# EPICS IOC start-up script: iocBoot/iocxxx/examples/vme.iocsh
# BEGIN vme.cmd ---------------------------------------------------------------

### Scalers: Joerger VSC8/16
#dbLoadRecords("$(SCALER)/db/scaler.db","P=$(PREFIX),S=scaler2,OUT=#C1 S0 @,DTYP=Joerger VSC8/16,FREQ=10000000")
#- scaler database with modified calcs (user calcs for all 16 channels)
dbLoadRecords("$(SCALER)/db/scaler16m.db","P=$(PREFIX),S=scaler1,OUT=#C0 S0 @,DTYP=Joerger VSC8/16,FREQ=10000000")
#- Joerger VSC setup parameters:
#-     (1)cards, (2)base address(ext, 256-byte boundary),
#-     (3)interrupt vector (0=disable or  64 - 255)
VSCSetup(2, 0xB0000000, 200)

#- Joerger VS
#- scalerVS_Setup(int num_cards, /* maximum number of cards in crate */
#-       char *addrs,            /* address (0x800-0xf800, 2048-byte (0x800) boundary) */
#-       unsigned vector,        /* valid vectors(64-255) */
#-       int intlevel)
#scalerVS_Setup(1, 0x2000, 205, 5)
#epicsEnvSet("devScaler_VSDebug", 0)
#dbLoadRecords("$(STD)/stdApp/Db/scaler16m.db","P=$(PREFIX),S=scaler3,OUT=#C0 S0 @, DTYP=Joerger VS, FREQ=10000000")

# Heidenhain IK320 VME encoder interpolator
#dbLoadRecords("$(VME)/vmeApp/Db/IK320card.db","P=$(PREFIX),sw2=card0:,axis=1,switches=41344,irq=3")
#dbLoadRecords("$(VME)/vmeApp/Db/IK320card.db","P=$(PREFIX),sw2=card0:,axis=2,switches=41344,irq=3")
#dbLoadRecords("$(VME)/vmeApp/Db/IK320group.db","P=$(PREFIX),group=5")

# Struck 3801 MCS setup. mca 7-3-1
#< st_SIS3801.iocsh

# Struck 3820 MCS setup. mca 7-3-1
#< st_SIS3820.iocsh

#- VMI4116 setup parameters:
#-     (1)cards, (2)base address(short, 36-byte boundary),
#devAoVMI4116Debug = 20
#VMI4116_setup(1, 0xff00)
#dbLoadRecords("$(VME)/vmeApp/Db/VME_DAC.db", "P=$(PREFIX),D=2,C=0,N=1,S=0,DTYP=VMIVME-4116,H=65536,L=0", std)
#dbLoadRecords("$(VME)/vmeApp/Db/VME_DAC.db", "P=$(PREFIX),D=2,C=0,N=2,S=1,DTYP=VMIVME-4116,H=65536,L=0", std)
#dbLoadRecords("$(VME)/vmeApp/Db/VME_DAC.db", "P=$(PREFIX),D=2,C=0,N=3,S=2,DTYP=VMIVME-4116,H=65536,L=0", std)
#dbLoadRecords("$(VME)/vmeApp/Db/VME_DAC.db", "P=$(PREFIX),D=2,C=0,N=4,S=3,DTYP=VMIVME-4116,H=65536,L=0", std)
#dbLoadRecords("$(VME)/vmeApp/Db/VME_DAC.db", "P=$(PREFIX),D=2,C=0,N=5,S=4,DTYP=VMIVME-4116,H=65536,L=0", std)
#dbLoadRecords("$(VME)/vmeApp/Db/VME_DAC.db", "P=$(PREFIX),D=2,C=0,N=6,S=5,DTYP=VMIVME-4116,H=65536,L=0", std)
#dbLoadRecords("$(VME)/vmeApp/Db/VME_DAC.db", "P=$(PREFIX),D=2,C=0,N=7,S=6,DTYP=VMIVME-4116,H=65536,L=0", std)
#dbLoadRecords("$(VME)/vmeApp/Db/VME_DAC.db", "P=$(PREFIX),D=2,C=0,N=8,S=7,DTYP=VMIVME-4116,H=65536,L=0", std)

# vme test record
dbLoadRecords("$(VME)/vmeApp/Db/vme.db", "P=$(PREFIX),Q=vme1")

# Hewlett-Packard 10895A Laser Axis (interferometer)
#iocshLoad("$(VME)/iocsh/HP_10895A.iocsh", "PREFIX=$(PREFIX), MAX_CARDS=2, ADDRESS=0x1000, INSTANCE=HPLaser1, CARD=0")
#iocshLoad("$(VME)/iocsh/HP_10895A.iocsh", "PREFIX=$(PREFIX), INSTANCE=HPLaser2, CARD=1")

# Acromag general purpose Digital I/O
#iocshLoad("$(VME)/iocsh/Acromag_AVME9440.iocsh", "PREFIX=$(PREFIX), MAX_CARDS=2, ADDRESS=0x0400, INT_VEC=0x78, INSTANCE=1, CARD=0")
#iocshLoad("$(VME)/iocsh/Acromag_AVME9440.iocsh", "PREFIX=$(PREFIX), INSTANCE=2, CARD=1")

# Bunch-clock generator
#iocshLoad("$(VME)/iocsh/BunchClkGen.iocsh", "PREFIX=$(PREFIX), INSTANCE=1, CARD=0, ADDRESS=0x8c00")

### GP307 Vacuum Controller
#dbLoadRecords("$(VME)/vmeApp/Db/gp307.db","P=$(PREFIX)")

# Machine Status Link (MSL) board (MRD 100)
#iocshLoad("$(VME)/iocsh/MSL_MRD100.iocsh", "PREFIX=$(PREFIX), INSTANCE=01, ADDRESS=0xB0000200, INT_VEC=0xA0, CARD=0")

# Allen-Bradley 6008 scanner
#abConfigNlinks(1)
#abConfigVme(0,0xc00000,0x60,5)
#abConfigAuto()

# APS quad electrometer
#< quadEM.cmd

# END vme.cmd -----------------------------------------------------------------
